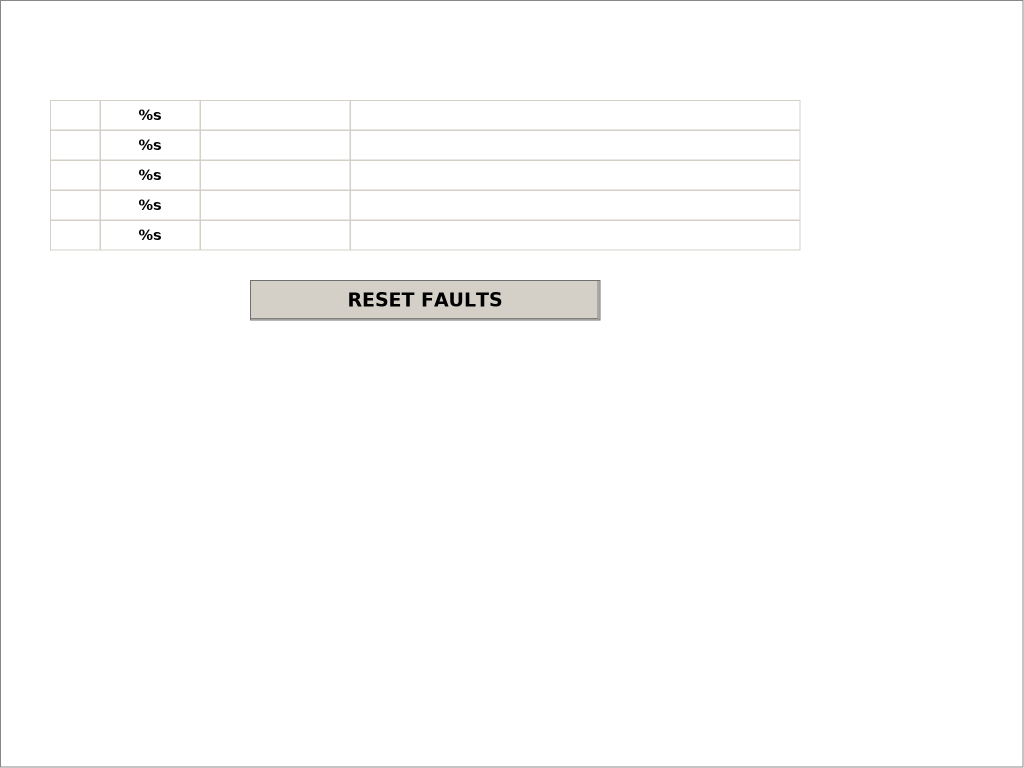
VISUALIZATION MessageScreen  // 1024x768
    Group (50,100 750x220)
        Group (0,0 750x30)
            Textfield (0,0 50x30), text list: 'E_FaultTypes', text index: IBF_Utilities.GVL_Message.arActiveFaults[0].FaultType
            Textfield (50,0 100x30), "%s", text variable: IBF_Utilities.GVL_Message.arActiveFaults[0].FullFaultId
            Textfield (150,0 150x30), text list: 'E_Locations', text index: IBF_Utilities.GVL_Message.arActiveFaults[0].LocationNumber
            Textfield (300,0 450x30), text list: 'TL_MessageDiscriptions', text index: IBF_Utilities.GVL_Message.arActiveFaults[0].MessageNumber
        Group (0,30 750x30)
            Textfield (0,0 50x30), text list: 'E_FaultTypes', text index: IBF_Utilities.GVL_Message.arActiveFaults[1].FaultType
            Textfield (50,0 100x30), "%s", text variable: IBF_Utilities.GVL_Message.arActiveFaults[1].FullFaultId
            Textfield (150,0 150x30), text list: 'E_Locations', text index: IBF_Utilities.GVL_Message.arActiveFaults[1].LocationNumber
            Textfield (300,0 450x30), text list: 'TL_MessageDiscriptions', text index: IBF_Utilities.GVL_Message.arActiveFaults[1].MessageNumber
        Group (0,60 750x30)
            Textfield (0,0 50x30), text list: 'E_FaultTypes', text index: IBF_Utilities.GVL_Message.arActiveFaults[2].FaultType
            Textfield (50,0 100x30), "%s", text variable: IBF_Utilities.GVL_Message.arActiveFaults[2].FullFaultId
            Textfield (150,0 150x30), text list: 'E_Locations', text index: IBF_Utilities.GVL_Message.arActiveFaults[2].LocationNumber
            Textfield (300,0 450x30), text list: 'TL_MessageDiscriptions', text index: IBF_Utilities.GVL_Message.arActiveFaults[2].MessageNumber
        Group (0,90 750x30)
            Textfield (0,0 50x30), text list: 'E_FaultTypes', text index: IBF_Utilities.GVL_Message.arActiveFaults[3].FaultType
            Textfield (50,0 100x30), "%s", text variable: IBF_Utilities.GVL_Message.arActiveFaults[3].FullFaultId
            Textfield (150,0 150x30), text list: 'E_Locations', text index: IBF_Utilities.GVL_Message.arActiveFaults[3].LocationNumber
            Textfield (300,0 450x30), text list: 'TL_MessageDiscriptions', text index: IBF_Utilities.GVL_Message.arActiveFaults[3].MessageNumber
        Group (0,120 750x30)
            Textfield (0,0 50x30), text list: 'E_FaultTypes', text index: IBF_Utilities.GVL_Message.arActiveFaults[4].FaultType
            Textfield (50,0 100x30), "%s", text variable: IBF_Utilities.GVL_Message.arActiveFaults[4].FullFaultId
            Textfield (150,0 150x30), text list: 'E_Locations', text index: IBF_Utilities.GVL_Message.arActiveFaults[4].LocationNumber
            Textfield (300,0 450x30), text list: 'TL_MessageDiscriptions', text index: IBF_Utilities.GVL_Message.arActiveFaults[4].MessageNumber
        Button (200,180 350x40), "RESET FAULTS"
            tap IBF_Utilities.GVL_Message.bResetFaults
END_VISUALIZATION

(* stored: Version 1.1.0.1, ProductVersion 3.1.4024.9
   Visu MessageScreen: Id {b97efdc7-02af-4e74-98ce-29826f21ef34} *)
